// TIA Portal V16 export
// export: Created 2021-07-12T14:47:18.6777433Z, ExportSetting WithDefaults, DisplayName Totally Integrated Automation Portal, DisplayVersion V16, DisplayName TIA Portal Version Control Interface, DisplayVersion V16, DisplayName TIA Portal Openness, DisplayVersion V16, DisplayName STEP 7 Professional, DisplayVersion V16, DisplayName STEP 7 Safety, DisplayVersion V16, DisplayName WinCC Professional, DisplayVersion V16
TYPE "LSimaHydTO_typeValveCharacteristic"
TITLE = LSimaHydTO_typeValveCharacteristic
// Valve characteristic
// stored: IsFailsafeCompliant false
   STRUCT
      DB_NUMBER { S7_SetPoint := 'True'} : UInt;   // Number of DB of type LSimaHydTO_typeVCharData with valve profile data
      SmoothChangeTime { S7_SetPoint := 'True'} : Real;   // Filter time for smooth changing
      SmoothingMode { S7_SetPoint := 'True'} : Int;   // Filter mode for smooth changing: 0: T1 / 1: ramping with constant ramp / 2: ramping with time
   END_STRUCT;
END_TYPE
